Universal Robots PolyScope program: nut_l2r.urp

Program nut_l2r (installation=default directory=/programs/phev_demos createdIn=5.9.1.1031110 lastSavedIn=5.9.1.1031110 robotSerialNumber=20195501059)
Calibrated DH parameters: a=[0.000146, -0.418764, -0.053981, 0.000058, -0.000023, 0]; d=[0.162545, 37.319448, -206.067439, 168.881546, 0.09955, 0.099464]; alpha=[1.57004, -0.001979, 0.002304, 1.570607, -1.57066, 0]; deltaTheta=[0, -0.174616, -1.258233, 1.432844, -0.000001, 0]
BeforeStart
  start_p := get_actual_tcp_pose()
  MoveJ speed 60 deg/s, acceleration 80 deg/s^2 (useActiveTCP=true) feature=Base
    Waypoint Waypoint (Variable): variable(name=start_p)
  Call safe_home
Robot Program (runOnlyOnce=true)
  Loop Forever
    MoveL speed 250 mm/s, acceleration 1200 mm/s^2 (useActiveTCP=true) feature=Base
      Waypoint Waypoint (Variable): variable(featureName=i01_NutStackL)
    Call pick_nut
    URCap Grip Check (Robotiq_Grippers, Robotiq Inc.) dataModel(ObjectDetectedKey=true, GripperIdKey=1, ModelDefinedKey=true, DimensionKey=76.73962608299132, DimensionNegativeGapKey=2.070223438212494, DimensionDimensionPositiveGapKey=2.070223438212494, DimensionValidationKey=false); state(isChildrenLocked=true)
      URCap If (Robotiq_Grippers, Robotiq Inc.)
        MoveL speed 250 mm/s, acceleration 1200 mm/s^2 (useActiveTCP=true) feature=Base
          Waypoint Waypoint (Variable): variable(featureName=i01_NutStackR)
        Call drop_nut
      URCap Else (Robotiq_Grippers, Robotiq Inc.)
        MoveL speed 250 mm/s, acceleration 1200 mm/s^2 (useActiveTCP=true) feature=Base
          URCap Gripper (Robotiq_Grippers, Robotiq Inc.) dataModel(position=100.0, force=100.0, speed=100.0, positionInDouble=100.0, forceInDouble=100.0, speedInDouble=100.0, slaveIds=[9], blocking=false)
          Waypoint Waypoint (Variable): variable(featureName=i01_Home)
        Halt
SubProgram  [hidden by the author, left out]
SubProgram  [hidden by the author, left out]
SubProgram  [hidden by the author, left out]
SubProgram safe_home [hidden by the author, left out]
SubProgram pick_nut [hidden by the author, left out]
SubProgram drop_nut [hidden by the author, left out]
